// TIA Portal V20 export
DATA_BLOCK "DB82-OPOUT"   // DB82
{ S7_Optimized_Access := 'FALSE' }
// stored: AutoNumber false
   VAR
      L001 : Bool;   // L001-T1A - Mod Operare Manual Selectat
      L002 : Bool;   // L002-T1A - Mod Operare Automat Selectat
      L003 : Bool;   // L003-T1A - Aruncator - In Pozitia "Sus"
      L004 : Bool;   // L004-T1A - Aruncator - In Pozitia "Jos"
      L005 : Bool;   // L005-T1A - Aruncator 1 - Teava Prezenta
      L006 : Bool;   // L006-T1A - Aruncator 2 - Teava Prezenta
      L007 : Bool;   // L007-T1A - CaleRole - Senzor 1 - Teava Prezenta
      L008 : Bool;   // L008-T1A - CaleRole - Senzor 2 - Teava Prezenta
      L009 : Bool;   // L009-T1A - Lant (transport) - In Pozitia "Pas"
      L010 : Bool;   // L010-T1A - Senzor Start Masurare Lungime Teava
      L011 : Bool;   // L011-T1A - CaleRole - Rotire Inainte
      L012 : Bool;   // L012-T1A - CaleRole - Rotire Inapoi
      L013 : Bool;   // L013-T1A - Pipe Ident
      L014 : Bool;
      L015 : Bool;   // L015-T1A - Lant (transport) - Deplasare Inainte
      L016 : Bool;   // L016-T1A - Lant (transport) - Deplasare Inapoi
      L017 : Bool;   // L017-T1A - Opritor - Deplasare Inainte
      L018 : Bool;   // L018-T1A - Opritor - Deplasare Inapoi
      L019 : Bool;   // L019-Pompa 1 Regim Auto/Manual
      L020 : Bool;   // L020-T1A - Lant (transport) - Pas Efectuat
      L021 : Bool;   // L021-T1A - Incarcare Blocata
      L022 : Bool;   // L022-T1A - Control Pupitru Local
      L023 : Bool;   // L023-T1C - Control Pupitru Cabina
      L024 : Bool;   // L024-T1C - Control Pupitru Local
      L025 : Bool;   // L025-T1C - Mod Operare Manual Selectat
      L026 : Bool;   // L026-T1C - Mod Operare Automat Selectat
      L027 : Bool;   // L027-T1C - Aruncator - In Pozitia "Sus"
      L028 : Bool;   // L028-T1C - Aruncator - In Pozitia "Jos"
      L029 : Bool;   // L029-T1C - Aruncator 1 - Teava Prezenta
      L030 : Bool;   // L030-T1C - Aruncator 2 - Teava Prezenta
      L031 : Bool;   // L031-T1C - CaleRole - Senzor 1 - Teava Prezenta
      L032 : Bool;   // L032-T1C - CaleRole - Senzor 2 - Teava Prezenta
      L033 : Bool;   // L033-T1C - CaleRole - Senzor 3 - Teava Prezenta
      L034 : Bool;   // L034-T1C - Senzor Start Masurare Lungime Teava
      L035 : Bool;   // L035-T1C - Lant (transport) - In Pozitia "Pas"
      L036 : Bool;   // L036-T1C - Lant (transport) - Deplasare Inainte
      L037 : Bool;   // L037-T1C - Lant (transport) - Deplasare Inapoi
      L038 : Bool;   // L038-T1C - Pipe Ident
      L039 : Bool;
      L040 : Bool;   // L040-T1C - CaleRole - Rotire Inainte
      L041 : Bool;   // L041-T1C - CaleRole - Rotire Inapoi
      L042 : Bool;   // L042-T1C - Opritor - Deplasare Inainte
      L043 : Bool;   // L043-T1C - Opritor - Deplasare Inapoi
      L044 : Bool;
      L045 : Bool;   // L045-T1A - Scuturator comandat
      L046 : Bool;   // L046-T1C - Incarcare Blocata
      L047 : Bool;   // L047-T1C - Scuturator comandat
      L048 : Bool;   // L048-T1A - Control Pupitru Cabina
      L049 : Bool;   // L049-T1A - Lant - Mod Operare Pas
      L050 : Bool;   // L050-T1A - Lant - Mod Operare Continuu
      L051 : Bool;   // L051-T1C - Lant - Mod Operare Pas
      L052 : Bool;   // L052-T1C - Lant - Mod Operare Continuu
      L053 : Bool;   // L053-T4 - Lant - Mod Operare Pas
      L054 : Bool;   // L054-T4 - Lant - Mod Operare Continuu
      L055 : Bool;   // L055-T5 - Lant - Mod Operare Pas
      L056 : Bool;   // L056-T5 - Lant - Mod Operare Continuu
      L057 : Bool;   // L057-T4 - Mod Operare Manual Selectat
      L058 : Bool;   // L058-T4 - Mod Operare Automat Selectat
      L059 : Bool;   // L059-T4 - CaleRole 1 - Rotire Inainte
      L060 : Bool;   // L060-T4 - CaleRole 1 - Rotire Inapoi
      L061 : Bool;   // L061-T4 - CaleRole 2 - Rotire Inainte
      L062 : Bool;   // L062-T4 - CaleRole 2 - Rotire Inapoi
      L063 : Bool;   // L063-T4 - Excentric - Rotire Inainte
      L064 : Bool;   // L064-T3 - CaleRole - Senzor - Teava Prezenta
      L065 : Bool;   // L065-T4 - Opritor - In Pozitia "Sus"
      L066 : Bool;   // L066-T4 - Opritor - In Pozitia "Jos"
      L067 : Bool;   // L067-T4 - Lant (transport) - Deplasare Inainte
      L068 : Bool;   // L068-T4 - Lant (transport) - Deplasare Inapoi
      L069 : Bool;   // L069-T4 - Lant (rostogolire) - Deplasare Inainte
      L070 : Bool;   // L070-T4 - Lant (rostogolire) - Deplasare Inapoi
      L071 : Bool;   // L071-T4 - Lant (transport) - Pas Efectuat
      L072 : Bool;   // L072-T4 - CaleRole 1 - Senzor 1 - Teava Prezenta
      L073 : Bool;   // L073-T4 - CaleRole 1 - Senzor 2 - Teava Prezenta
      L074 : Bool;   // L074-T4 - CaleRole 1 - Senzor 3 - Teava Prezenta
      L075 : Bool;   // L075-T4 - CaleRole 2 - Senzor 1 - Teava Prezenta
      L076 : Bool;   // L076-T4 - CaleRole 2 - Senzor 2 - Teava Prezenta
      L077 : Bool;   // L077-T4 - CaleRole 2 - Senzor 3 - Teava Prezenta
      L078 : Bool;   // L078-T4 - Excentric - In Pozitia "Initial"
      L079 : Bool;   // L079-T4 - Excentric - In Pozitia "Vertical"
      L080 : Bool;   // L080-T4 - Intrare Lant - Senzor 1 - Teava Prezenta
      L081 : Bool;   // L081-T4 - Intrare Lant - Senzor 2 - Teava Prezenta
      L082 : Bool;   // L082-T4 - Iesire Lant - Senzor 1 - Teava Prezenta
      L083 : Bool;   // L083-T4 - Iesire Lant - Senzor 2 - Teava Prezenta
      L084 : Bool;   // Calea cu role T4.1 senzor 4 suplimentar
      L085 : Bool;   // L085-T4 - Excentric Rotire Blocata
      L086 : Bool;   // L086-T4 - Descarcare Blocata
      L087 : Bool;   // L087-T6 - Lant - Mod Operare Pas
      L088 : Bool;   // L088-T6 - Lant - Mod Operare Continuu
      L089 : Bool;   // L089-T7A - Lant - Mod Operare Pas
      L090 : Bool;   // L090-T7A - Lant - Mod Operare Continuu
      L091 : Bool;   // L091-T7B - Lant - Mod Operare Pas
      L092 : Bool;   // L092-T7B - Lant - Mod Operare Continuu
      L093 : Bool;   // L093-T4 - Iesire Lant - Senzor 1 (incetinire) - Teava Prezenta
      L094 : Bool;   // L094-T4 - Iesire Lant - Senzor 2 (incetinire) - Teava Prezenta
      L095 : Bool;   // L095-T4 - Iesire Lant - (ultima pozitie in tracking) - Teava Prezenta
      L096 : Bool;   // L096-T4 - Iesire Lant - (ultima pozitie in tracking) - Teava Prezenta
      L097 : Bool;   // L097-T5 - Mod Operare Manual Selectat
      L098 : Bool;   // L098-T5 - Mod Operare Automat Selectat
      L099 : Bool;   // L099-T5 - CaleRole 1 - Rotire Inainte
      L100 : Bool;   // L100-T5 - CaleRole 1 - Rotire Inapoi
      L101 : Bool;   // L101-T5 - CaleRole 2 - Rotire Inainte
      L102 : Bool;   // L102-T5 - CaleRole 2 - Rotire Inapoi
      L103 : Bool;   // L103-T5 - Excentric - Rotire Inainte
      L104 : Bool;   // L104-T5 - Descarcare Blocata
      L105 : Bool;   // L105-T5 - Excentric - In Pozitia "Initial"
      L106 : Bool;   // L106-T5 - Excentric - In Pozitia "Vertical"
      L107 : Bool;   // L107-T5 - Lant (rostogolire) - Deplasare Inainte
      L108 : Bool;   // L108-T5 - Lant (rostogolire) - Deplasare Inapoi
      L109 : Bool;   // L109-T5 - Lant (transport) - Deplasare Inainte
      L110 : Bool;   // L110-T5 - Lant (transport) - Deplasare Inapoi
      L111 : Bool;   // L111-T5 - Lant (transport) - Pas Efectuat
      L112 : Bool;   // L112-T5 - Opritor - In Pozitia "Sus"
      L113 : Bool;   // L113-T5 - Opritor - In Pozitia "Jos"
      L114 : Bool;   // L114-T5 - CaleRole 1 - Senzor 1 - Teava Prezenta
      L115 : Bool;   // L115-T5 - CaleRole 1 - Senzor 2 - Teava Prezenta
      L116 : Bool;   // L116-T5 - CaleRole 2 - Senzor 1 - Teava Prezenta
      L117 : Bool;   // L117-T5 - CaleRole 2 - Senzor 2 - Teava Prezenta
      L118 : Bool;   // L118-T5 - CaleRole 2 - Senzor 3 Intrare Cuptor - Teava Prezenta
      L119 : Bool;   // L119-T5 - Intrare Lant - Senzor 1 - Teava Prezenta
      L120 : Bool;   // L120-T5 - Intrare Lant - Senzor 2 - Teava Prezenta
      L121 : Bool;   // L121-T5 - Iesire Lant - Senzor 1 - Teava Prezenta
      L122 : Bool;   // L122-T5 - Iesire Lant - Senzor 2 - Teava Prezenta
      L123 : Bool;   // L123-T5 - Excentric - Rotire Inapoi
      L124 : Bool;   // L124-T5 - Iesire Lant - Senzor 1 (incetinire) - Teava Prezenta
      L125 : Bool;   // L125-T5 - Iesire Lant - Senzor 2 (incetinire) - Teava Prezenta
      L126 : Bool;   // L126-T5 - Iesire Lant - (ultima pozitie in tracking) - Teava Prezenta
      L127 : Bool;   // L127-T5 - Iesire Lant - (ultime pozitie in tracking) - Teava Prezenta
      L128 : Bool;
      L129 : Bool;   // L129-Taiere Probe - Manual
      L130 : Bool;   // L130-Taiere Probe - Automat
      L131 : Bool;
      L132 : Bool;
      L133 : Bool;
      L134 : Bool;
      L135 : Bool;
      L136 : Bool;
      L137 : Bool;   // L137-T1E - Mod Operare Manual Selectat
      L138 : Bool;   // L138-T1E - Mod Operare Automat Selectat
      L139 : Bool;   // L139-T1E - Aruncator - In Pozitia "Sus"
      L140 : Bool;   // L140-T1E - Aruncator - In Pozitia "Jos"
      L141 : Bool;   // L141-T1E - Dozator Tevi - In Pozitia "Sus"
      L142 : Bool;   // L142-T1E - Dozator Tevi - In Pozitia "Jos"
      L143 : Bool;   // L143-T1E - Aruncator - Senzor 1 - Teava Prezenta
      L144 : Bool;   // L144-T1E - Aruncator - Senzor 2 - Teava Prezenta
      L145 : Bool;   // L145-T1E - Dozator Tevi - Senzor 1 - Teava Prezenta
      L146 : Bool;   // L146-T1E - Dozator Tevi - Senzor 1 - Teava Prezenta
      L147 : Bool;
      L148 : Bool;   // L148-T1E - Opritor - Deplasare Inainte
      L149 : Bool;   // L149-T1E - Opritor - Deplasare Inapoi
      L150 : Bool;
      L151 : Bool;
      L152 : Bool;   // L152 - Indicatie "Oprire de Urgenta" Actionata in Zona 1
      L153 : Bool;   // L153 - Indicatie "Oprire de Urgenta" Actionata in Zona 2
      L154 : Bool;   // L154 - Indicatie "Oprire de Urgenta" Actionata in Zona 3
      L155 : Bool;   // L155 - Indicatie "Oprire de Urgenta" Actionata in Zona 4
      L156 : Bool;   // L156 - Indicatie "Oprire de Urgenta" Actionata in Zona 5
      L157 : Bool;   // L157 - Indicatie "Oprire de Urgenta" Actionata in Zona 6
      L158 : Bool;   // L158 - Indicatie "Oprire de Urgenta" Actionata in Zona 7
      L159 : Bool;   // L159 - Indicatie "Oprire de Urgenta" Actionata in Zona 8
      L160 : Bool;
      L161 : Bool;   // L161- LM4 - Control Pupitru Cabina
      L162 : Bool;   // L162- LM4 - Control Pupitru Local
      L163 : Bool;   // L163- LM5 - Control Pupitru Cabina
      L164 : Bool;   // L164- LM5 - Control Pupitru Local
      L165 : Bool;   // L165- LM6 - Control Pupitru Cabina
      L166 : Bool;   // L166- LM6 - Control Pupitru Local
      L167 : Bool;   // L167- LM7 - Control Pupitru Cabina
      L168 : Bool;   // L168- LM7 - Control Pupitru Local
      L169 : Bool;   // L169-T6 - Mod Operare Manual Selectat
      L170 : Bool;   // L170-T6 - Mod Operare Automat Selectat
      L171 : Bool;   // L171-T6 - Excentric - Rotire Inainte
      L172 : Bool;   // L172-T6 - Descarcare Blocata
      L173 : Bool;   // L173-T6 - Excentric - Rotire Inapoi
      L174 : Bool;   // L174-T6 - Excentric - In Pozitia "Initial"
      L175 : Bool;   // L175-T6 - Excentric - In Pozitia "Vertical"
      L176 : Bool;   // L176-T6 - CaleRole - Rotire Inainte
      L177 : Bool;   // L177-T6 - CaleRole - Rotire Inapoi
      L178 : Bool;   // L178-T6 - Opritor - In Pozitia "Sus"
      L179 : Bool;   // L179-T6 - Opritor - In Pozitia "Jos"
      L180 : Bool;   // L180-T6 - Lant (transport) - Deplasare Inainte
      L181 : Bool;   // L181-T6 - Lant (transport) - Deplasare Inapoi
      L182 : Bool;   // L182-T6 - Lant (transport) - Pas Efectuat
      L183 : Bool;   // L183-T6 - Intrare Lant - Senzor 1 - Teava Prezenta
      L184 : Bool;   // L184-T6 - Intrare Lant - Senzor 2 - Teava Prezenta
      L185 : Bool;   // L185-T6 - Iesire Lant - Senzor 1 - Teava Prezenta
      L186 : Bool;   // L186-T6 - Iesire LAnt - Senzor 2 - Teava Prezenta
      L187 : Bool;   // L187-T6 - CaleRole - Senzor 1 - Teava Prezenta
      L188 : Bool;   // L188-T6 - CaleRole - Senzor 2 - Teava Prezenta
      L189 : Bool;   // L189-T6 - Senzor Start Masurare Lungime Teava
      L190 : Bool;   // L190-T6 - Excentric Rotire Blocata
      L191 : Bool;   // L191-T6 - Iesire Lant - Senzor 1 (incetinire) - Teava Prezenta
      L192 : Bool;   // L192-T6 - Iesire Lant - Senzor 2 (incetinire) - Teava Prezenta
      L193 : Bool;   // L193-T6 - Iesire Lant - (ultima pozitie in tracking) - Teava Prezenta
      L194 : Bool;   // L194-T6 - Iesire Lant - (ultima pozitie in tracking) - Teava Prezenta
      L195 : Bool;   // L195-T6 - Iesire Lant - (ultima pozitie in tracking) - Teava Prezenta
      L196 : Bool;   // L195-T6 - Intrare lant - Senzor mijloc -Teava prezenta
      L197 : Bool;
      L198 : Bool;   // L198-T4 - Lant - Alarma Tracking
      L199 : Bool;   // L199-T5 - Lant - Alarma Tracking
      L200 : Bool;   // L100-T6 - Lant - Alarma Tracking
      L201 : Bool;   // L201-T1D - Mod Operare Manual Selectat
      L202 : Bool;   // L202-T1D - Mod Operare Automat Selectat
      L203 : Bool;   // L203-T1D - Aruncator - In Pozitia "Sus"
      L204 : Bool;   // L204-T1D - Aruncator - In Pozitia "Jos"
      L205 : Bool;   // L205-T1D - Opritor - Deplasare Inainte
      L206 : Bool;   // L206-T1D - Opritor - Deplasare Inapoi
      L207 : Bool;   // L207-T1D - Pipe Ident
      L208 : Bool;   // L208-T1D - CaleRole - Rotire Inainte
      L209 : Bool;   // L209-T1D - CaleRole - Rotire Inapoi
      L210 : Bool;   // L210-T1D - Aruncator - Senzor 1 - Teava Prezenta
      L211 : Bool;   // L211-T1D - Aruncator - Senzor 2 - Teava Prezenta
      L212 : Bool;   // L212-T1D - CaleRole - Senzor 1 - Teava Prezenta
      L213 : Bool;   // L213-T1D - CaleRole - Senzor 2 - Teava Prezenta
      L214 : Bool;   // L214-T1D - Senzor Start Masurare Lungime Teava
      L215 : Bool;   // L215-T1D - Incarcare Blocata
      L216 : Bool;
      L217 : Bool;
      L218 : Bool;
      L219 : Bool;
      L220 : Bool;   // T6 - Senzor 3 incetinire lant
      L221 : Bool;   // T6 - Senzor 4 ultima pozitie banca lant
      L222 : Bool;   // T6 - Senzor 4 pe calea cu role
      L223 : Bool;
      L224 : Bool;
      L225 : Bool;   // L225-T7 - Mod Operare Manual Selectat
      L226 : Bool;   // L226-T7 - Mod Operare Automat Selectat
      L227 : Bool;   // L227-T7 - CaleRole - Rotire Inainte
      L228 : Bool;   // L228-T7 - CaleRole - Rotire Inapoi
      L229 : Bool;   // L229-T7 - Aruncator - In Pozitia "Sus"
      L230 : Bool;   // L230-T7 - Aruncator - In Pozitia "Jos"
      L231 : Bool;   // L231-T7 - Excentric 1 - Rotire Inainte
      L232 : Bool;   // L232-T7 - Excentric 1 - Rotire Inapoi
      L233 : Bool;
      L234 : Bool;   // L234-T7 - Excentric 1 - In Pozitia "Vertical"
      L235 : Bool;   // L235-T7 - Excentric 1 - In Pozitia "Initial"
      L236 : Bool;   // L236-T7 - Excentric 2 - Rotire Inainte
      L237 : Bool;   // L237-T7 - Excentric 2 - Rotire Inapoi
      L238 : Bool;
      L239 : Bool;   // L239-T7 - Excentric 2 - In Pozitia "Vertical"
      L240 : Bool;   // L240-T7 - Excentric 2 - In Pozitia "Initial"
      L241 : Bool;   // L241-T7 - Excentric 1 - Senzor 1 - Teava Prezenta
      L242 : Bool;   // L242-T7 - Excentric 1 - Senzor 2 - Teava Prezenta
      L243 : Bool;   // L243-T7 - Excentric 2 - Senzor 1 - Teava Prezenta
      L244 : Bool;   // L244-T7 - Excentric 2 - Senzor 2 - Teava Prezenta
      L245 : Bool;   // L245-T7 - CaleRole - Senzor 1 - Teava Prezenta
      L246 : Bool;   // L246-T7 - CaleRole - Senzor 2 - Teava Prezenta
      L247 : Bool;   // L247-T7 - CaleRole - Senzor 3 - Teava Prezenta
      L248 : Bool;
      L249 : Bool;
      L250 : Bool;   // L250-T4 - Aliniere Teava - Cap
      L251 : Bool;   // L251-T4 - Aliniere Teava - Coada
      L252 : Bool;
      L253 : Bool;
      L254 : Bool;   // Alarma posibil teava blocata in calitor
      L255 : Bool;   // Eroare comunicatie cu Level2 (Teava Nemarcata)
      L256 : Bool;   // L256-Apa - Control Pupitru Cabina
      L257 : Bool;   // L257-T7A - Mod Operare Manual Selectat
      L258 : Bool;   // L258-T7A - Mod Operare Automat Selectat
      L259 : Bool;   // L259-T7A - CaleRole - Rotire Inainte
      L260 : Bool;   // L260-T7A - CaleRole - Rotire Ianpoi
      L261 : Bool;   // L261-T7A - Excentric 1 - Rotire Inainte
      L262 : Bool;   // L261-T7A - Descarcare Blocata
      L263 : Bool;   // L263-T7A - Excentric 1 - Rotire Inapoi
      L264 : Bool;   // L264-T7A - Excentric 1 - In Pozitia "Vertical"
      L265 : Bool;   // L265-T7A - Excentric 1 - In Pozitia "Initial"
      L266 : Bool;   // L266-T7A - Excentric 2 - Rotire Inainte
      L267 : Bool;   // L266-T7A - Excentric 2 - Rotire Inapoi
      L268 : Bool;   // Senzor mijloc lant iesire T7A
      L269 : Bool;   // L269-T7A - Excentric 1 - In Pozitia "Initial"
      L270 : Bool;   // L270-T7A - Excentric 1 - In Pozitia "Vertical"
      L271 : Bool;   // L271-T7A - Lant (rostogolire) - Deplasare Inainte
      L272 : Bool;   // L272-T7A - Lant (rostogolire) - Deplasare Inapoi
      L273 : Bool;   // L273-T7A - Lant (transport) - Deplasare Inainte
      L274 : Bool;   // L274-T7A - Lant (transport) - Deplasare Inapoi
      L275 : Bool;   // L275-T7A - Lant (transport) - Pas Efectuat
      L276 : Bool;   // L276-T7A - Excentric 1 - Senzor 1 - Teava Prezenta
      L277 : Bool;   // L277-T7A - Excentric 1 - Senzor 2 - Teava Prezenta
      L278 : Bool;   // L278-T7A - Intrare Lant - Senzor 1 - Teava Prezenta
      L279 : Bool;   // L279-T7A - Intrare Lant - Senzor 2 - Teava Prezenta
      L280 : Bool;   // L280-T7A - Iesire Lant - Senzor 1 - Teava Prezenta
      L281 : Bool;   // L281-T7A - Iesire Lant - Senzor 2 - Teava Prezenta
      L282 : Bool;   // L282-T7A - CaleRole - Senzor 1 - Teava Prezenta
      L283 : Bool;   // L283-T7A - CaleRole - Senzor 2 - Teava Prezenta
      L284 : Bool;   // L284-T7A - CaleRole - Senzor 3 - Teava Prezenta
      L285 : Bool;   // L285-T7AB - Masina Marcare - Senzor (inainte de marcare) - Teava Prezenta
      L286 : Bool;   // L286-T7AB - Masina Marcare - Senzor (dupa de marcare) - Teava Prezenta
      L287 : Bool;   // L287-T7AB - Masina Marcare - Senzor - In Pozitia "Ridicat"
      L288 : Bool;   // L288-T7AB - Masina Marcare - Senzor - In Pozitia "Coborat" (cu teava prezenta)
      L289 : Bool;   // L289-T7AB - Masina Marcare - ElectroElectroValva Ridicare
      L290 : Bool;   // L290-T7AB - Masina Marcare - ElectroElectroValva Coborare
      L291 : Bool;   // L291-T7AB - Masina Marcare - Marcare Pornita
      L292 : Bool;   // L292-T7AB - Masina Marcare - Mod Operare Automat
      L293 : Bool;   // L293-T7AB - Masina Marcare - Mod Operare Manual
      L294 : Bool;   // L294-T7AB - Masina Marcare - Dezactivata
      L295 : Bool;   // L295-T7AB - Masina Marcare - Vopsea Marcare OK
      L296 : Bool;   // L296-T7AB - Masina Marcare - Pompa OK
      L297 : Bool;   // L297-T7B - Mod Operare Manual Selectat
      L298 : Bool;   // L298-T7B - Mod Operare Automat Selectat
      L299 : Bool;   // L299-T7B - CaleRole - Rotire Inainte
      L300 : Bool;   // L300-T7B - CaleRole - Rotire Inapoi
      L301 : Bool;   // L301-T7B - Lant Colector - Deplasare Urcare
      L302 : Bool;   // L302-T7B - Lant Colector - Deplasare Coborare
      L303 : Bool;   // L303-T7B - Aruncator 1 - In Pozitia "Sus"
      L304 : Bool;   // L304-T7B - Aruncator 1 - In Pozitia "Jos"
      L305 : Bool;   // L305-T7B - Aruncator 2 - In Pozitia "Sus"
      L306 : Bool;   // L306-T7B - Aruncator 2 - In Pozitia "Jos"
      L307 : Bool;   // L307-T7B - Aruncator 1 - Senzor 1 - Teava Prezenta
      L308 : Bool;   // L308-T7B - Aruncator 1 - Senzor 2 - Teava Prezenta
      L309 : Bool;   // L309-T7B - Aruncator 2 - Senzor 1 - Teava Prezenta
      L310 : Bool;   // L310-T7B - Aruncator 2 - Senzor 2 - Teava Prezenta
      L311 : Bool;   // L311-T7B - CaleRole - Senzor 1 - Teava Prezenta
      L312 : Bool;   // L312-T7B - CaleRole - Senzor 2 - Teava Prezenta
      L313 : Bool;   // L313-T7B - CaleRole - Senzor 3 - Teava Prezenta
      L314 : Bool;   // L314-T7B - Lant Colector - In Pozitia "Sus"
      L315 : Bool;   // L315-T7B - Lant Colector - In Pozitia "Jos"
      L316 : Bool;   // L316-T7B - Lant (rostogolire) - Deplasare Inainte
      L317 : Bool;   // L317-T7B - Lant (rostogolire) - Deplasare Inapoi
      L318 : Bool;   // L319-T7B - Lant (transport) - Deplasare Inapoi
      L319 : Bool;   // L318-T7B - Lant (transport) - Deplasare Inainte
      L320 : Bool;   // L320-T7B - Lant (transport) - Pas Efectuat
      L321 : Bool;   // L321-T7B - Intrare Lant - Senzor 1 - Teava Prezenta
      L322 : Bool;   // L322-T7B - Intrare Lant - Senzor 2 - Teava Prezenta
      L323 : Bool;   // L323-T7B - Iesire Lant - Senzor 1 - Teava Prezenta
      L324 : Bool;   // L324-T7B - Iesire Lant - Senzor 2 - Teava Prezenta
      L325 : Bool;   // L325-T7B - Lant Colector - Senzor 1 - Plin
      L326 : Bool;   // L326-T7B - Lant Colector - Senzor 2 - Plin
      L327 : Bool;   // L327-T3 - Deztunderizator Activat
      L328 : Bool;   // L328-T3 - Deztunderizator Dezactivat
      L329 : Bool;   // L329-T3 - CaleRole - Rotire Inainte
      L330 : Bool;   // L330-T3 - CaleRole - Rotire Inapoi
      L331 : Bool;   // L331-T3 - Cap Calitor 1 - Deplasare Ridicare
      L332 : Bool;   // L332-T3 - Cap Calitor 1 - Deplasare Coborare
      L333 : Bool;   // L333-T3 - Cap Calitor 2 - Deplasare Ridicare
      L334 : Bool;   // L334-T3 - Cap Calitor 2 - Deplasare Coborare
      L335 : Bool;   // L335-T3 - Cap Calitor 3 - Deplasare Ridicare
      L336 : Bool;   // L336-T3 - Cap Calitor 3 - Deplasare Coborare
      L337 : Bool;   // L337-T3 - Grinda - Deplasare Ridicare
      L338 : Bool;   // L338-T3 - Grinda - Deplasare Coborare
      L339 : Bool;   // L339-T3 - Filtru - Rotire Inainte
      L340 : Bool;   // L340-T3 - Filtru - Rotire Inapoi
      L341 : Bool;   // L341-T3 - ServoElectroValva Filtru - Activata
      L342 : Bool;   // L341-T3 - ServoElectroValva Filtru - Dezactivata
      L343 : Bool;   // L343-T3 - Servovalva Stropire - Activata
      L344 : Bool;
      L345 : Bool;   // L345-T7C - Mod Operare Manual Selectat
      L346 : Bool;   // L346-T7C - Mod Operare Automat Selectat
      L347 : Bool;   // L347-T7C - CaleRole - Rotire Inainte
      L348 : Bool;   // L348-T7C - CaleRole - Rotire Inapoi
      L349 : Bool;   // L349-T7C - Lant Colector - Deplasare Ridicare
      L350 : Bool;   // L350-T7C - Lant Colector - Deplasare Coborare
      L351 : Bool;   // L351-T7C - Aruncator - In Pozitia "Sus"
      L352 : Bool;   // L352-T7C - Aruncator - In Pozitia "Jos"
      L353 : Bool;   // L353-T7C - CaleRole - Senzor 1 - Teava Prezenta
      L354 : Bool;   // L354-T7C - CaleRole - Senzor 2 - Teava Prezenta
      L355 : Bool;   // L355-T7C - CaleRole - Senzor 3 - Teava Prezenta
      L356 : Bool;   // L356-T7C - Lant Colector - In Pozitia "Sus"
      L357 : Bool;   // L357-T7C - Lant Colector - In Pozitia "Jos"
      L358 : Bool;   // L358-T7C - Opritor Mobil - Deplasare Sus
      L359 : Bool;   // L359-T7C - Opritor Mobil - Deplasare Jos
      L360 : Bool;   // L360-T7C - Opritor Mobil - In Pozitia "Sus"
      L361 : Bool;   // L361-T7C - Opritor Mobil - In Pozitia "Jos"
      L362 : Bool;   // L362-T7C - Prelevare ContraProbe Abilitata
      L363 : Bool;   // L363-T7C - CaleRole - Deplasare Sus
      L364 : Bool;   // L364-T7C - CaleRole - Deplasare Jos
      L365 : Bool;
      L366 : Bool;
      L367 : Bool;
      L368 : Bool;
      L369 : Bool;
      L370 : Bool;   // L370-Apa - Mod Operare Manual Selectat
      L371 : Bool;   // L371-Apa - Mod Operare Automat Selectat
      L372 : Bool;
      L373 : Bool;
      L374 : Bool;   // L374-Apa - Cel Putin 1 Alarma Activa
      L375 : Bool;   // L375-Apa - Pompa 1 (pompa principala) - Pornita
      L376 : Bool;   // L376-Apa - Pompa 1 (pompa principala) - Oprita
      L377 : Bool;   // L377-Apa - Pompa 2 (pompa principala) - Pornita
      L378 : Bool;   // L378-Apa - Pompa 2 (pompa principala) - Oprita
      L379 : Bool;   // L379-Apa - Pompa 3 (pompa principala) - Pornita
      L380 : Bool;   // L380-Apa - Pompa 1 (pompa principala) - Oprita
      L381 : Bool;   // L381-Apa - Pompa 4 (pompa principala) - Pornita
      L382 : Bool;   // L382-Apa - Pompa 4 (pompa principala) - Oprita
      L383 : Bool;   // L383-Apa - Pompa 5 (pompa turnuri racire) - Pornita
      L384 : Bool;   // L384-Apa - Pompa 5 (pompa turnuri racire) - Oprita
      L385 : Bool;   // L385-Apa - Pompa 5R - Pornita
      L386 : Bool;   // L386-Apa - Pompa 5R - Oprita
      L387 : Bool;   // L387-Apa - Pompa 5 Selectata
      L388 : Bool;   // L388-Apa - Pompa 5R Selectata
      L389 : Bool;   // L389-Apa - Pompa 8 (pompa drenaj) - Pornita
      L390 : Bool;   // L390-Apa - Pompa 8 (pompa drenaj) - Oprita
      L391 : Bool;   // L391-Apa - Pompa 9 (pompa tunder) - Pornita
      L392 : Bool;   // L392-Apa - Pompa 9 (pompa tunder) - Oprita
      L393 : Bool;   // L393-Apa - Pompa 10 (pompa evacuare canal) - Pornita
      L394 : Bool;   // L394-Apa - Pompa 10 (pompa evacuare canal) - Oprita
      L395 : Bool;   // L395-Apa - Pompa 11 (pompa evacuare avarie) - Pornita
      L396 : Bool;   // L396-Apa - Pompa 11 (pompa evacuare avarie) - Oprita
      L397 : Bool;   // L397-Apa - Pompa Rez - Pornita
      L398 : Bool;   // L398-Apa - Pompa Rez - Oprita
      L399 : Bool;   // Ventilator 3 racire cuplat
      L400 : Bool;   // L400-Apa - Transportator Elicoidal TE1 - Pornit
      L401 : Bool;   // L401-Apa - Transportator Elicoidal TE1 - Oprit
      L402 : Bool;   // L402-Apa - Transportator Elicoidal TE2 - Pornit
      L403 : Bool;   // L403-Apa - Transportator Elicoidal TE1 - Oprit
      L404 : Bool;   // L404-Apa - Semnalizare Selectie/Deselectie Deztunderizator
      L405 : Bool;   // L405-Apa - Semnalizare Selectie/Deselectie Cap Calitor
      L406 : Bool;   // L406-Apa - Ventilator Turn Racire 1 - Pornit
      L407 : Bool;   // L407-Apa - Ventilator Turn Racire 1 - Oprit
      L408 : Bool;   // L408-Apa - Ventilator Turn Racire 2 - Pornit
      L409 : Bool;   // L409-Apa - Ventilator Turn Racire 2 - Oprit
      L410 : Bool;   // L410-Apa - Deztunderizator SIKO - Pornit
      L411 : Bool;   // Ventilator 4 racire cuplat
      L412 : Bool;   // L412-Apa - ElectroValva Y1 - Actionat Directia 1
      L413 : Bool;   // L413-Apa - ElectroValva Y1 - Actionat Directia 2
      L414 : Bool;   // L414-Apa - ElectroValva Y2 - Actionat Directia 1
      L415 : Bool;   // L415-Apa - ElectroValva Y2 - Actionat Directia 2
      L416 : Bool;   // L416-Apa - ElectroValva Y3 - Actionat Directia 1
      L417 : Bool;   // L417-Apa - ElectroValva Y3 - Actionat Directia 2
      L418 : Bool;
      L419 : Bool;   // L419-Apa - Pompa 1 Selectata
      L420 : Bool;   // L420-Apa - Pompa 2 Selectata
      L421 : Bool;   // L421-Apa - Pompa 3 Selectata
      L422 : Bool;   // L422-Apa - Pompa 4 Selectata
      L423 : Bool;   // L423-Apa - Pompa Rez Selectata
      L424 : Bool;
      L425 : Bool;   // L425-Apa - Ventilator Turn Racire 1 - Rotire Turatie Mica
      L426 : Bool;   // L426-Apa - Ventilator Turn Racire 1 - Rotire Turatie Mare
      L427 : Bool;   // L427-Apa - Ventilator Turn Racire 2 - Rotire Turatie Mica
      L428 : Bool;   // L428-Apa - Ventilator Turn Racire 1 - Rotire Turatie Mare
      L429 : Bool;
      L430 : Bool;
      L431 : Bool;   // L431-Apa - Pompa 1 - Sesizor Curgere
      L432 : Bool;   // L432-Apa - Pompa 2 - Sesizor Curgere
      L433 : Bool;   // L433-Apa - Pompa 3 - Sesizor Curgere
      L434 : Bool;   // L434-Apa - Pompa 4 - Sesizor Curgere
      L435 : Bool;   // L435-Apa - Pompa 5 - Sesizor Curgere
      L436 : Bool;   // L436-Apa - Pompa 5R - Sesizor Curgere
      L437 : Bool;   // L437-Apa - Pompa 7 - Sesizor Curgere
      L438 : Bool;   // L438-Apa - Pompa 8 - Sesizor Curgere
      L439 : Bool;   // L439-Apa - Pompa 9 - Sesizor Curgere
      L440 : Bool;   // L440-Apa - Pompa 10 - Sesizor Curgere
      L441 : Bool;   // L441-Apa - Pompa 11 - Sesizor Curgere
      L442 : Bool;   // L442-Apa - Bazin Tunder - Senzor Nivel Maxim
      L443 : Bool;   // L443-Apa - Bazin Tunder - Senzor Nivel Minim
      L444 : Bool;   // L444-Apa - Bazin Pompare - Senzor Nivel Maxim
      L445 : Bool;   // L445-Apa - Bazin Pompare - Senzor Nivel Minim
      L446 : Bool;   // L446-Apa - Racitor Pornit
      L447 : Bool;   // L447-Apa - Instalatie Depozitare Pornita
      L448 : Bool;   // L448-Apa - Filtru Autocuratate FA2 Pornit
      L449 : Bool;   // L449-Apa - Senzor Presiune scazuta pe Linia de Calire
      L450 : Bool;   // L450-Apa - Senzor Presiune Scazuta Turnuri Racire
      L451 : Bool;
      L452 : Bool;
      L453 : Bool;   // L453-Apa - Control Pupitru Local Apa
      L454 : Bool;
      L455 : Bool;   // L455-T3 - Cap Calitor 1 - Deplasare Sus
      L456 : Bool;   // L456-T3 - Cap Calitor 1 - Deplasare Jos
      L457 : Bool;   // L457-T3 - Cap Calitor 2 - Deplasare Sus
      L458 : Bool;   // L458-T3 - Cap Calitor 2 - Deplasare Jos
      L459 : Bool;   // L459-T3 - Cap Calitor 3 - Deplasare Sus
      L460 : Bool;   // L460-T3 - Cap Calitor 3 - Deplasare Jos
      L461 : Bool;   // L461-T3 - Grinda - Deplasare Sus
      L462 : Bool;   // L462-T3 - Grinda - Deplasare Jos
      L463 : Bool;   // L463- Deztunderizator - Mod Operare Automat Selectat
      L464 : Bool;   // L464- Deztunderizator - Mod Operare Manual Selectat
      L465 : Bool;   // L465-T7A - Mod Operare Manual Selectat
      L466 : Bool;   // L466-T7A - Mod Operare Automat Selectat
      L467 : Bool;   // L467-T7A - CaleRole - Rotire Inainte
      L468 : Bool;   // L468-T7A - CaleRole - Rotire Inapoi
      L469 : Bool;   // L469-T7A - Excentric 1 - Rotire Inapoi
      L470 : Bool;   // L470-T7A - Excentric 1 - In Pozitia "Vertical"
      L471 : Bool;   // L471-T7A - Excentric 1 - In Pozitia "Initial"
      L472 : Bool;   // L472-T7A - Excentric 2 - Rotire Inainte
      L473 : Bool;   // L473-T7A - Excentric 1 - In Pozitia "Initial"
      L474 : Bool;   // L474-T7A - Excentric 1 - In Pozitia "Vertical"
      L475 : Bool;   // L475-T7A - Lant (rostogolire) - Deplasare Inainte
      L476 : Bool;   // L476-T7A - Lant (rostogolire) - Deplasare Inapoi
      L477 : Bool;   // L477-T7A - Lant (transport) - Deplasare Inainte
      L478 : Bool;   // L478-T7A - Lant (transport) - Deplasare Inapoi
      L479 : Bool;   // L479-T7A - Lant (transport) - Pas Efectuat
      L480 : Bool;   // L480-T7A - Excentric 1 - Senzor 1 - Teava Prezenta
      L481 : Bool;   // L481-T7A - Excentric 1 - Senzor 2 - Teava Prezenta
      L482 : Bool;   // L482-T7A - Intrare Lant - Senzor 1 - Teava Prezenta
      L483 : Bool;   // L483-T7A - Intrare Lant - Senzor 2 - Teava Prezenta
      L484 : Bool;   // L484-T7A - Iesire Lant - Senzor 1 - Teava Prezenta
      L485 : Bool;   // L485-T7A - Iesire Lant - Senzor 2 - Teava Prezenta
      L486 : Bool;   // L486-T7A - CaleRole - Senzor 1 - Teava Prezenta
      L487 : Bool;   // L487-T7A - CaleRole - Senzor 2 - Teava Prezenta
      L488 : Bool;   // L488-T7A - CaleRole - Senzor 3 - Teava Prezenta
      L489 : Bool;
      L490 : Bool;   // Ventilator Turn 3 pornit
      L491 : Bool;   // Ventilator Turn 3 oprit
      L492 : Bool;   // Ventilator Turn 4 pornit
      L493 : Bool;   // Ventilator Turn 4 oprit
      L494 : Bool;
      L495 : Bool;
      L496 : Bool;
      L497 : Bool;   // L497-T7B - Mod Operare Manual Selectat
      L498 : Bool;   // L498-T7B - Mod Operare Automat Selectat
      L499 : Bool;   // L499-T7B - CaleRole - Rotire Inainte
      L500 : Bool;   // L500-T7B - CaleRole - Rotire Inapoi
      L501 : Bool;   // L501-T7B - Lant Colector - Deplasare Sus
      L502 : Bool;   // L502-T7B - Lant Colector - Deplasare Jos
      L503 : Bool;   // L503-T7B - Aruncator 1 - In Pozitia "Sus"
      L504 : Bool;   // L504-T7B - Aruncator 1 - In Pozitia "Jos"
      L505 : Bool;   // L505-T7B - Aruncator 2 - In Pozitia "Sus"
      L506 : Bool;   // L506-T7B - Aruncator 2 - In Pozitia "Jos"
      L507 : Bool;   // L507-T7B - Aruncator 1 - Senzor 1 - Teava Prezenta
      L508 : Bool;   // L508-T7B - Aruncator 1 - Senzor 2 - Teava Prezenta
      L509 : Bool;   // L509-T7B - Aruncator 2 - Senzor 1 - Teava Prezenta
      L510 : Bool;   // L510-T7B - Aruncator 2 - Senzor 2 - Teava Prezenta
      L511 : Bool;   // L511-T7B - CaleRole - Senzor 1 - Teava Prezenta
      L512 : Bool;   // L512-T7B - CaleRole - Senzor 2 - Teava Prezenta
      L513 : Bool;   // L513-T7B - CaleRole - Senzor 3 - Teava Prezenta
      L514 : Bool;   // L514-T7B - Lant Colector - In Pozitia "Sus"
      L515 : Bool;   // L515-T7B - Lant Colector - In Pozitia "Jos"
      L516 : Bool;   // L516-T7B - Lant (rostogolire) - Deplasare Inainte
      L517 : Bool;   // L517-T7B - Lant (rostogolire) - Deplasare Inapoi
      L518 : Bool;   // L518-T7B - Lant (transport) - Deplasare Inainte
      L519 : Bool;   // L519-T7B - Lant (transport) - Deplasare Inapoi
      L520 : Bool;   // L520-T7B - Lant (transport) - Pas Efectuat
      L521 : Bool;   // L521-T7B - Intrare Lant - Senzor 1 - Teava Prezenta
      L522 : Bool;   // L522-T7B - Intrare Lant - Senzor 2 - Teava Prezenta
      L523 : Bool;   // L523-T7B - Iesire Lant - Senzor 1 - Teava Prezenta
      L524 : Bool;   // L524-T7B - Iesire Lant - Senzor 2 - Teava Prezenta
      L525 : Bool;   // L525-T7B - Lant Colector - Senzor 1 - Plin
      L526 : Bool;   // L526-T7B - Lant colector - Senzor 2 - Plin
      L527 : Bool;
      L528 : Bool;
      L529 : Bool;
      L530 : Bool;
      L531 : Bool;
      L532 : Bool;
      L533 : Bool;
      L534 : Bool;
      L535 : Bool;
      L536 : Bool;
      L537 : Bool;   // L537-T7C - Mod Operare Manual Selectat
      L538 : Bool;   // L538-T7C - Mod Operare Automat Selectat
      L539 : Bool;   // L539-T7C - CaleRole - Rotire Inainte
      L540 : Bool;   // L540-T7C - CaleRole - Rotire Inapoi
      L541 : Bool;   // L541-T7C - Lant Colector - Deplasare Sus
      L542 : Bool;   // L542-T7C - Lant Colector - Deplasare Jos
      L543 : Bool;   // L543-T7C - Aruncator - In Pozitia "Sus"
      L544 : Bool;   // L544-T7C - Aruncator - In Pozitia "Jos"
      L545 : Bool;   // L545-T7C - CaleRole - Senzor 1 - Teava Prezenta
      L546 : Bool;   // L546-T7C - CaleRole - Senzor 2 - Teava Prezenta
      L547 : Bool;   // L547-T7C - CaleRole - Senzor 3 - Teava Prezenta
      L548 : Bool;   // L548-T7C - Lant Colector - In Pozitia "Sus"
      L549 : Bool;   // L549-T7C - Lant Colector - In Pozitia "Jos"
      L550 : Bool;   // L550-T7C - Opritor Mobil - Deplasare Sus
      L551 : Bool;   // L551-T7C - Opritor Mobil - Deplasare Jos
      L552 : Bool;   // L552-T7C - Opritor Mobil - Deplasare Sus
      L553 : Bool;   // L553-T7C - Opritor Mobil - Deplasare Jos
      L554 : Bool;
      L555 : Bool;
      L556 : Bool;
      L557 : Bool;
      L558 : Bool;
      L559 : Bool;
      L560 : Bool;
      L561 : Bool;   // L560-L370-Apa - Mod Operare Manual Selectat
      L562 : Bool;   // L561-L371-Apa - Mod Operare Automat Selectat
      L563 : Bool;
      L564 : Bool;
      L565 : Bool;
      L566 : Bool;
      L567 : Bool;
      L568 : Bool;
      L569 : Bool;   // L569-T7C - Debitare - Masina DezAbilitata
      L570 : Bool;   // L569-T7C - Debitare - Role T7C - In Pozitia 'Ridicat'
      L571 : Bool;   // L569-T7C - Debitare - Role T7C - In Pozitia 'Coborit'
      L572 : Bool;   // L569-T7C - Debitare - Opritor Mobil - Miscare 'Ridicare'
      L573 : Bool;   // L569-T7C - Debitare - Opritor Mobil - Miscare 'Coborire'
      L574 : Bool;   // L569-T7C - Debitare - Opritor Mobil - in Pozitia 'Ridicat'
      L575 : Bool;   // L569-T7C - Debitare - Opritor Mobil - in Pozitia 'Coborit'
      L576 : Bool;   // L569-T7C - Debitare - Menghina - Miscare 'Stringere'
      L577 : Bool;   // L569-T7C - Debitare - Menghina - Miscare 'Deschidere'
      L578 : Bool;   // L569-T7C - Debitare - Menghina - in Pozitia 'Inchis'
      L579 : Bool;   // L569-T7C - Debitare - Menghina - in Pozitia 'Deschis'
      L580 : Bool;   // L569-T7C - Debitare - Lama Circulara - Miscare 'Ridicare'
      L581 : Bool;   // L569-T7C - Debitare - Lama Circulara - Miscare 'Coborire'
      L582 : Bool;   // L569-T7C - Debitare - Lama Circulara - Ridicata
      L583 : Bool;   // L569-T7C - Debitare - Lama Circulara - Coborita
      L584 : Bool;   // L569-T7C - Debitare - Lama Circulara - Miscare 'Rotire'
      L585 : Bool;   // L569-T7C - Debitare - Lama Circulara - Convertizor 'Avarie'
      L586 : Bool;   // L569-T7C - Debitare - Temperatura Minima Ulei Hidraulic (start incalzire)
      L587 : Bool;   // L569-T7C - Debitare - Temperatura Ridicata Ulei Hidraulic (start ventilatie)
      L588 : Bool;   // L569-T7C - Debitare - Temperatura Maxima Ulei Hidraulic
      L589 : Bool;   // L569-T7C - Debitare - Nivel Minim Ulei Hidraulic
      L590 : Bool;   // L569-T7C - Debitare - Pompa Hidraulica Pornita
      L591 : Bool;   // L569-T7C - Debitare - Incalzire Pornita
      L592 : Bool;   // L569-T7C - Debitare - Ventilatie Pornita
      L593 : Bool;   // L569-T7C - Debitare - Nivel Minim Apa
      L594 : Bool;   // L569-T7C - Debitare - Pompa Apa Racire Pornita
      L595 : Bool;   // L569-T7C - Debitare - Lubrifiere Lama Pornita
      L596 : Bool;
      L597 : Bool;
      L598 : Bool;
      L599 : Bool;   // L599-T3 - Unitate 200bar selectata_PSC
      L600 : Bool;   // L600-T3 - Unitate 100bar selectata
      L601 : Bool;   // L601-T3 - Unitate 180bar selectata
      L602 : Bool;   // L602-T3 - Pompa joasa presiune 9.1 selectata
      L603 : Bool;   // L603-T3 - Pompa joasa presiune 9.2 selectata
      L604 : Bool;   // L604-T3 - Pompa joasa presiune pornita
      L605 : Bool;   // L605-T3 - Pompa inalta presiune pornita
      L606 : Bool;   // L606-T3 - Presostat apa alimentare
      L607 : Bool;   // L607-T3 - Senzor proximitate Robinet izolare 6.1 inainte pompa 9.2
      L608 : Bool;   // L608-T3 - Senzor proximitate Robinet izolare 6.2 inainte pompa 9.1
      L609 : Bool;   // L609-T3 - Senzor proximitate Robinet izolare 6.3 dupa pompa 9.2
      L610 : Bool;   // L610-T3 - Senzor proximitate Robinet izolare 6.4 dupa pompa 9.1
      L611 : Bool;   // L611-T3 - Robinet pneumatic Inalta presiune 20.1 deschis
      L612 : Bool;   // L612-T3 - Robinet pneumatic 29.2 deschis
      L613 : Bool;   // L613-T3 - Robinet pneumatic 29.1 deschis
      L614 : Bool;   // L614-t3 -Robinet sinclercolins 29.1 selectat
      L615 : Bool;   // L615-T3 -Robinet sinclercolins 29.1 selectat
      L616 : Bool;   // L603-T3 - Pompa joasa presiune 9.3 selectata
      L617 : Bool;   // Fierastrau Kasto: Emergency
      L618 : Bool;   // Fierastrau Kasto: Ready
      L619 : Bool;   // Fierastrau Kasto: Taiere pornita
      L620 : Bool;   // Fierastrau Kasto: Taiere Terminata
      L621 : Bool;   // Fierastrau Kasto: Avarie/avertizare
      L622 : Bool;   // Role Kasto: Prezenta teava intrare
      L623 : Bool;   // Fierastrau Kasto: Local/Distanta 1 = distanta
      L624 : Bool;   // L603-T3 - Pompa joasa presiune 9.4 selectata
      L625 : Bool;   // Role Kasto - Deplasare Inainte
      L626 : Bool;   // Role Kasto - Deplasare Inapoi
      L627 : Bool;   // Role Kasto: Prezenta teava pe role nr. 3
      L628 : Bool;   // Role Kasto: Prezenta teava pe role nr. 6
      L629 : Bool;   // Role Kasto: Prezenta teava pe role nr. 9
      L630 : Bool;   // Role Kasto: Prezenta teava pe role nr. 11
      L631 : Bool;   // Role Kasto: Prezenta teava pe role nr. 13
      L632 : Bool;   // Role Kasto: Prezenta teava inainte de rola mobila
      L633 : Bool;   // Role Kasto: Prezenta teava dupa rola mobila inainte Kasto
      L634 : Bool;   // Role Kasto: Prezenta teava in Kasto (la tampon)
      L635 : Bool;
      L636 : Bool;
      L637 : Bool;   // Marcare: Limita cursa sus motomartinet
      L638 : Bool;   // Marcare: Limita cursa jos motomartinet
      L639 : Bool;   // Marcare: Senzor de ZERO cursa motomartinet
      L640 : Bool;   // Marcare: Brat Marcare nu este sus
      L641 : Bool;   // Marcare: Senzor Marcare Cap
      L642 : Bool;   // Rola centrare cap refulat: Proximitate ridicata
      L643 : Bool;   // Rola centrare cap refulat: Proximitate coborata
      L644 : Bool;   // Tampon masurare proba: Limita cursa inainte
      L645 : Bool;   // Tampon masurare proba: Limita cursa inapoi
      L646 : Bool;   // Alarma zona Kasto
      L647 : Bool;   // Activare taiere teava cu cap refulat
      L648 : Bool;
      L649 : Bool;   // PompaRacire1 - Avarie Convertizor
      L650 : Bool;   // PompaRacire1 - Limita Curent Convertizor
      L651 : Bool;   // PompaRacire1 - Suprasarcina Convertizor
      L652 : Bool;
      L653 : Bool;
      L654 : Bool;
      L655 : Bool;
      L656 : Bool;
      OCV_CONV_RST : Bool;   // OCV - Reset Convertizor
      OCV_CONV_HOME : Bool;   // OCV - Home Convertizor
      OCV_LED_ON : Bool;   // OCV - LED On
      OCV_LED_OFF : Bool;   // OCV - LED Off
      OCV_CAM_START : Bool;   // OCV - Start Camera
      OCV_MOVE_UP : Bool;   // OCV - Comanda Ridicare
      OCV_MOVE_DW : Bool;   // OCV - Comanda Coborare
      OCV_AXAFESTO_HOME : Bool;   // OCV - Axa Festo Pozitie Home
      OCV_AXAFESTO_EME : Bool;   // OCV - Axa Festo in Emergenta [1=ok]
      OCV_AXAFESTO_SAFESTOP : Bool;   // OCV - Axa Festo Stop Safety
      OCV_AXAFESTO_DRVENA : Bool;   // OCV - Axa Festo Abilitare Convertizor
      OCV_ELECTROCV_COMM_OK : Bool;   // OCV - Electronica OCV Comunicatie OK
      OCV_ELECTROCV_READ_PROG : Bool;   // OCV - Electronica OCV Citire in Curs
      OCV_ELECTROCV_READ_DONE : Bool;   // OCV - Electronica OCV Citire Terminata
      OCV_MOVE_FBK_UP_POS : Bool;   // OCV - Confirmare Pozitie Ridicat
      OCV_MOVE_FBK_DW_POS : Bool;   // OCV - Confirmare Pozitie Coborat
      OCV_MOVE_ELE_TRIP : Bool;   // OCV - Avarie Deplasare
      OCV_MOVE_FBK_UP_Moving : Bool;   // OCV - Confirmare Deplasare Ridicare
      OCV_MOVE_FBK_DW_Moving : Bool;   // OCV - Confirmare Deplasare Coborare
      OCV_CLEAN_CMD_ON : Bool;   // OCV - Comanda Curatare Cap Marcare
      OCV_PURGE_CMD_ON : Bool;   // OCV - Comanda Purjare Cap Marcare
      OCV_CLEAN_CNT_ON : Bool;   // OCV - Indicatie Contorizare Timp Start Spray
      OCV_CLEAN_EXP_ON : Bool;   // OCV - Indicatie Timp Start Spray Depasit
      OCV_CLEAN_NIV_OK : Bool;   // OCV - Indicatie Nivel OK Solvent
      OCV_CLEAN_NIV_MIN : Bool;   // OCV - Indicatie Nivel Minim Solvent
      OCV_CLEAN_SLV_VLV : Bool;   // OCV - Indicatie Cap Marcare Valva Solvent
      OCV_START_MARCARE_CAP : Bool;   // OCV - Indicatie Prezenta Teava Start Marcare Cap
      OCV_START_MARCARE_COADA : Bool;   // OCV - Indicatie Prezenta Teava Start Marcare Coada
      bool_var : Array[0..56] of Int;
   END_VAR
BEGIN
END_DATA_BLOCK
